FUNCTION F_ChillerLoop_Error : FB_ChillerLoop
VAR_INPUT
END_VAR
VAR
	fbChillerLoop : FB_ChillerLoop;
END_VAR

fbChillerLoop(bLoopTempSW := FALSE);
F_ChillerLoop_Error := fbChillerLoop;

END_FUNCTION

(* stored: Version 1.1.0.1, ProductVersion 3.1.4022.17
   POU F_ChillerLoop_Error: Id {ac90e556-3ac2-46f7-b5b4-d1accc224a4f}, SpecialFunc None *)
